(* CoDeSys 2.3 export: D7TLINEST.EXP *)

(* Data type in D7Timer *)
TYPE D7TLineST :    (*структура одной линии расписания 7дн таймера*)
STRUCT
    wTimeOfWeek:    WORD;    (*время недели в минутах, к этому времени надо нагреть*)
    byTemp:         BYTE;    (*поддерживаемая температура*)
    byDur:          BYTE;    (*продолжительность в часах*)
END_STRUCT
END_TYPE
